FUNCTION_BLOCK FB_DefaultInputExample

VAR	
	// Default values of VAR_INPUT
	test, result1, result2 : INT;
END_VAR

// Fully defined input
result1 := M_Addition(input1 := test, input2 := 20);

// On required field declared, input2 has a default value of 25
result2 := M_Addition(input1 := test);

METHOD M_Addition :INT

VAR_INPUT
	input1 : INT;
	input2 : INT := 25;
END_VAR
M_Addition := input1 + input2;
END_METHOD

END_FUNCTION_BLOCK

(* stored: Version 1.1.0.1
   POU FB_DefaultInputExample: Id {73ec9b5b-fe84-46f8-9b10-6fe69d3f4155}, SpecialFunc None
   Method M_Addition: Id {cd3e7499-b676-47ad-9088-dd8fd204cb7b} *)
